TYPE IncrementalEncoderStatuses :
STRUCT
	///Is the device in a healthy state?
	healthStatus: HealthStatus;
	///Is the device in a busy state?
	busyStatus: BusyStatus;
END_STRUCT
END_TYPE

(* stored: Version 1.1.0.1, ProductVersion 3.1.4019.2
   DUT IncrementalEncoderStatuses: Id {b7bf7374-46e5-462e-8748-6678abfe5bc9} *)
